FUNCTION Deg2Rad : LREAL
VAR_INPUT
	deg: LREAL;
END_VAR
VAR
END_VAR

Deg2Rad := deg / 180.0 * PI;

END_FUNCTION

(* stored: Version 1.1.0.1, ProductVersion 3.1.4024.12
   POU Deg2Rad: Id {7b4aefb2-ead3-46ce-9e4e-ecd304a53f87}, SpecialFunc None *)
